PROGRAM Timer
VAR
	cnt	:	INT;
END_VAR

//Timer 1 ms
	GlobalVar.wMiliseconds := GlobalVar.wMiliseconds +1;
	IF GlobalVar.wMiliseconds >1000 THEN 
		GlobalVar.wMiliseconds := 0;
	END_IF

// Event Recorder
// Transmiting part of historian
cnt := cnt + 1;
IF cnt = 50 THEN
	cnt := 0;
	gvl.fbHistorian.Transmiting(HistorianDataPacket_EtherCAT => gvl.HistorianDataPacket_EtherCAT);		
	gvl.HistorianDataPacket_EtherCAT.TransmitRequest := gvl.fbHistorian.GetRequest;

END_IF

END_PROGRAM

(* stored: Version 1.1.0.1
   POU Timer: Id {2b7c21bf-c82f-47fb-b369-4bb9a5aa1a7f}, SpecialFunc None *)
